INTERFACE I_HMI

METHOD Buttons
VAR_INPUT
	bStart : BOOL;
	bStop : BOOL;
END_VAR
END_METHOD

METHOD Joystick
VAR_INPUT
	fJoyY : LREAL;
	fJoyX : LREAL;
END_VAR
END_METHOD

METHOD Lights
VAR_INPUT
	eLight : E_Light;
END_VAR
END_METHOD

METHOD ModeSelector
VAR_INPUT
	bAuto : BOOL;
	bManual : BOOL;
END_VAR
END_METHOD

END_INTERFACE

(* stored: Version 1.1.0.1, ProductVersion 3.1.4024.9
   Itf I_HMI: Id {251fceed-e838-489a-8a0d-24a86c22225d}
   Method Buttons: Id {24373131-a1ad-403d-b2b4-b32be369fc78}
   Method Joystick: Id {44924819-9d1f-4d07-b949-7eb3ff82412a}
   Method Lights: Id {e39e1801-c183-4146-aad9-50a124acbbbc}
   Method ModeSelector: Id {0fd1d885-6f37-46c1-a51e-05fd717f4a37} *)
